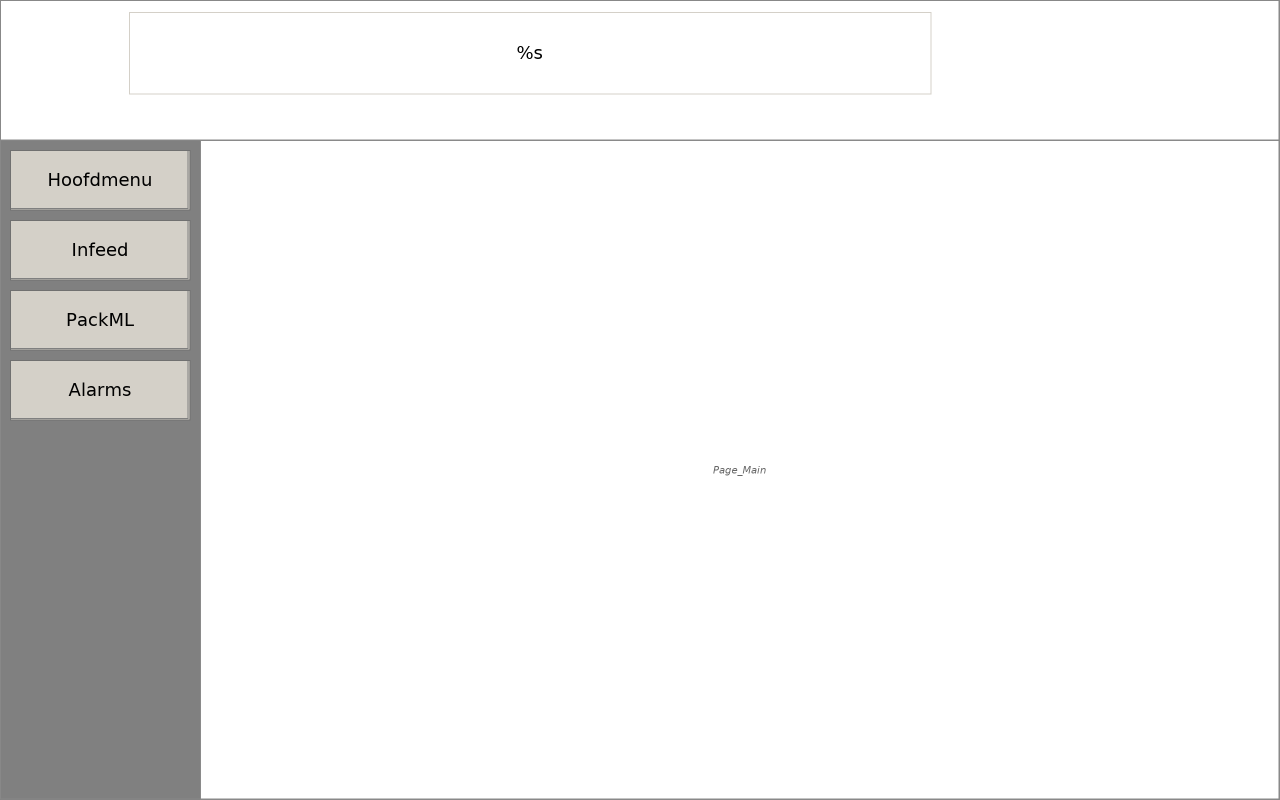
VISUALIZATION Visualization  // 1280x800
VAR_IN_OUT
END_VAR
VAR
	s_nPageIndex : DINT;
END_VAR
    Rectangle (0,140 200x660)
    Frame (0,0 1280x140)
        shows Header()
    Button (10,150 180x60), "Hoofdmenu", pressed state: s_nPageIndex = 0
        OnMouseClick: execute { s_nPageIndex := 0; }
    Button (10,220 180x60), "Infeed", pressed state: s_nPageIndex = 1
        OnMouseClick: execute { s_nPageIndex := 1; }
    Button (10,290 180x60), "PackML", pressed state: s_nPageIndex = 2
        OnMouseClick: execute { s_nPageIndex := 2; }
    Button (10,360 180x60), "Alarms", pressed state: s_nPageIndex = 3
        OnMouseClick: execute { s_nPageIndex := 3; }
    Frame (200,140 1080x660), frame switch variable: s_nPageIndex
        shows Page_Main()
        shows Page_Infeed()
        shows Page_PackML()
        shows Page_Alarms()
    Textfield (129,12 802x82), "%s", text variable: GVL_Modules.g_fbHmiAlarmList.q_sHighestActiveAlarm, colour toggle: GVL_Modules.g_unMachine.s_fbAlarmCollector.p_bStaRaised
        OnMouseClick: execute { s_npageIndex := 3; }
END_VISUALIZATION

(* stored: Version 1.1.0.1, ProductVersion 3.1.4026.13
   Visu Visualization: Id {8f3f86a6-4a57-4d7e-a731-0959e59203bc} *)
